Fanuc TP program (LS listing): MON_OP20L.LS

/PROG  MON_OP20L	  Cond
/ATTR
OWNER		= MNEDITOR;
COMMENT		= "";
PROG_SIZE	= 163;
CREATE		= DATE 20-02-06  TIME 22:57:46;
MODIFIED	= DATE 20-02-06  TIME 22:57:46;
FILE_NAME	= ;
VERSION		= 0;
LINE_COUNT	= 0;
MEMORY_SIZE	= 407;
PROTECT		= READ_WRITE;
TCD:  STACK_SIZE	= 0,
      TASK_PRIORITY	= 50,
      TIME_SLICE	= 0,
      BUSY_LAMP_OFF	= 0,
      ABORT_REQUEST	= 0,
      PAUSE_REQUEST	= 0;
DEFAULT_GROUP	= *,*,*,*,*;
CONTROL_CODE	= 00000000 00000000;
/APPL

AUTO_SINGULARITY_HEADER;
  ENABLE_SINGULARITY_AVOIDANCE   : TRUE;
/MN
/POS
/END
